PROGRAM MAIN
VAR	
END_VAR
VAR CONSTANT
END_VAR

// Only enable one example at a time. 
//-----------------------------------

POU_Example2PositionalMoves();
//POU_ExampleDynamicMoves();

END_PROGRAM

(* stored: Version 1.1.0.1, ProductVersion 3.1.4024.3
   POU MAIN: Id {852e9656-65ce-4dc2-8fb3-58084af07b1c}, SpecialFunc None *)
